(* IEC 61131-3 sources: Few-few/plc/src, 10 files *)

(* ---- DT_Tipi.st ---- *)
(*
 ============================================================================
   DT_Tipi.st  —  Tipi e enumerazioni comuni
   Software PLC manovra ascensore (geared / idraulico) — IEC 61131-3 ST
 ============================================================================
   NOTA DI SICUREZZA: questo software gestisce SOLO la logica di manovra.
   La catena di sicurezza e' cablata e indipendente (vedi schemi/).
 ============================================================================
*)

TYPE E_StatoMacchina :
(
    ST_RIPOSO       := 0,   (* cabina ferma a piano, porte chiuse *)
    ST_PRENOTATO    := 1,   (* chiamata acquisita, valuta partenza *)
    ST_CHIUDI_PORTE := 2,   (* chiusura porte prima della marcia   *)
    ST_PARTENZA     := 3,   (* sblocco freno / apertura valvola    *)
    ST_MARCIA       := 4,   (* marcia ad alta velocita'            *)
    ST_RALLENTA     := 5,   (* rallentamento verso il piano        *)
    ST_LIVELLA      := 6,   (* livellamento a bassa velocita'      *)
    ST_ARRESTO      := 7,   (* arresto e frenatura                 *)
    ST_APRI_PORTE   := 8,   (* apertura porte al piano             *)
    ST_ATTESA       := 9,   (* attesa con porte aperte             *)
    ST_REVISIONE    := 20,  (* modo ispezione uomo presente        *)
    ST_GUASTO       := 90,  (* fuori servizio per guasto           *)
    ST_EMERGENZA    := 91   (* catena sicurezza aperta             *)
) E_StatoMacchina;
END_TYPE

TYPE E_Direzione :
(
    DIR_FERMO  := 0,
    DIR_SALITA := 1,
    DIR_DISCESA := 2
) E_Direzione;
END_TYPE

(* Parametri configurabili (mappati su Modbus per il modulo WiFi).
   I valori safety-relevant (SR) restano protetti da chiave fisica. *)
TYPE ST_Parametri :
STRUCT
    (* --- non-safety (NS) --- *)
    TempoPorteAperte   : TIME := T#5S;    (* attesa porte aperte        *)
    TempoRichiusura    : TIME := T#3S;    (* dwell prima richiusura     *)
    NudgingAbilitato   : BOOL := TRUE;    (* richiusura forzata         *)
    TempoLuceOff       : TIME := T#120S;  (* spegnimento luce cabina    *)
    PianoParcheggio    : INT  := 0;       (* piano di sosta             *)
    RitardoParcheggio  : TIME := T#60S;
    GongAbilitato      : BOOL := TRUE;
    (* --- safety-relevant (SR) — modificabili solo con chiave fisica --- *)
    VelocitaIspezione  : REAL := 0.30;    (* m/s, <= 0.63 EN 81-20      *)
    VelocitaLivell     : REAL := 0.05;    (* m/s, <= 0.30               *)
    FinestraZonaPorta  : INT  := 35;      (* mm                         *)
    RelivellAbilitato  : BOOL := TRUE;
END_STRUCT
END_TYPE

(* Comandi calcolati dalla logica di posizionamento *)
TYPE ST_RichiestaCorsa :
STRUCT
    PianoTarget : INT := -1;     (* -1 = nessuna richiesta *)
    Direzione   : E_Direzione := DIR_FERMO;
    Valida      : BOOL := FALSE;
END_STRUCT
END_TYPE

(* ---- GVL_IO.st ---- *)
(*
 ============================================================================
   GVL_IO.st  —  Lista variabili globali / mappatura I/O fisica
   Software PLC manovra ascensore (geared / idraulico) — IEC 61131-3 ST
 ============================================================================
   Indirizzi %I / %Q indicativi per CPU Siemens S7-1200 1214C (DI14/DQ10)
   + moduli di espansione. Adattare alla configurazione reale.
   N. fermate di riferimento: 6 (piani 0..5).
 ============================================================================
*)

VAR_GLOBAL CONSTANT
    N_PIANI : INT := 6;   (* piani 0..5 *)
END_VAR

(* -------------------------- INGRESSI DIGITALI -------------------------- *)
VAR_GLOBAL
    (* sicurezza e modi *)
    xCatenaSicurezzaOK : BOOL AT %I0.0;   (* -KA-SIC feedback (1 = catena chiusa) *)
    xRevisione         : BOOL AT %I0.1;   (* -S-REV selettore revisione *)
    xRevSalita         : BOOL AT %I0.2;   (* -SB-REVU uomo presente su *)
    xRevDiscesa        : BOOL AT %I0.3;   (* -SB-REVD uomo presente giu *)

    (* posizione *)
    xZonaPorta1        : BOOL AT %I0.4;   (* -B-ZP1 *)
    xZonaPorta2        : BOOL AT %I0.5;   (* -B-ZP2 (ridondante) *)
    xRallentSalita     : BOOL AT %I0.6;   (* -B-RALL-U camma rallentamento su *)
    xRallentDiscesa    : BOOL AT %I0.7;   (* -B-RALL-D camma rallentamento giu *)
    xImpulsoPiano      : BOOL AT %I1.0;   (* -B-PIANI conteggio piani / encoder *)

    (* porte e carico *)
    xSovraccarico      : BOOL AT %I1.1;   (* -S-SOVR *)
    xFotocellula       : BOOL AT %I1.2;   (* -S-FOTO costa/barriera (1 = libero) *)
    xPortaAperta       : BOOL AT %I1.3;   (* -S-FAP finecorsa porta aperta *)
    xPortaChiusa       : BOOL AT %I1.4;   (* -S-FCP finecorsa porta chiusa *)

    (* protezioni macchina *)
    xTermicaMotore     : BOOL AT %I1.5;   (* -F-MOT 1 = ok *)
    xPressioneMin      : BOOL AT %I1.6;   (* -S-MINP solo idraulico, 1 = ok *)
    xControlloFreno    : BOOL AT %I1.7;   (* -S-FRE solo geared, 1 = freno integro *)

    (* chiamate cabina (parola, bit per piano) e chiamate piano *)
    wChiamateCabina    : WORD AT %IW2;    (* -SB-CAB-0..5 *)
    wChiamatePianoSu   : WORD AT %IW4;    (* -SB-PIA up   *)
    wChiamatePianoGiu  : WORD AT %IW6;    (* -SB-PIA down *)
END_VAR

(* --------------------------- USCITE DIGITALI -------------------------- *)
VAR_GLOBAL
    (* trazione geared *)
    xKM_Salita   : BOOL AT %Q0.0;   (* -KM-S *)
    xKM_Discesa  : BOOL AT %Q0.1;   (* -KM-D *)
    xKM_Veloce   : BOOL AT %Q0.2;   (* -KM-V alta velocita' (2V) *)
    xKM_Lento    : BOOL AT %Q0.3;   (* -KM-L bassa velocita' (2V) *)
    xKM_Freno    : BOOL AT %Q0.4;   (* -KM-FRE comando freno *)

    (* idraulico *)
    xKM_Pompa    : BOOL AT %Q0.5;   (* -KM-P linea pompa *)
    xKM_Stella   : BOOL AT %Q0.6;   (* -KM-Y *)
    xKM_Triangolo: BOOL AT %Q0.7;   (* -KM-Δ *)
    xEV_Salita   : BOOL AT %Q1.0;   (* -EV-S valvola salita *)
    xEV_Discesa  : BOOL AT %Q1.1;   (* -EV-D valvola discesa *)

    (* porte e segnalazioni *)
    xKM_ApriPorte  : BOOL AT %Q1.2; (* -KM-APRE *)
    xKM_ChiudiPorte: BOOL AT %Q1.3; (* -KM-CHIU *)
    xGong          : BOOL AT %Q1.4; (* -H-GONG *)
    xFuoriServizio : BOOL AT %Q1.5; (* -H-OOS *)
    wDisplayPos    : WORD AT %QW2;  (* -H-POS posizione cabina *)
    wFrecceDir     : WORD AT %QW4;  (* -H-DIR direzione *)
END_VAR

(* ------------------------- VARIABILI INTERNE -------------------------- *)
VAR_GLOBAL
    Par           : ST_Parametri;        (* parametri (anche via Modbus/WiFi) *)
    iPianoCorrente: INT := 0;            (* piano corrente stimato *)
    eDirezione    : E_Direzione := DIR_FERMO;
    eStato        : E_StatoMacchina := ST_RIPOSO;
    awChiamate    : ARRAY[0..5] OF BOOL; (* registro chiamate consolidato *)
END_VAR

(* ---- FC_Util.st ---- *)
(*
 ============================================================================
   FC_Util.st  —  Funzioni di utilita' per la mappatura Modbus dei parametri
 ============================================================================
   Conversioni registro<->valore scalato e secondi<->TIME.
   Usate da FB_ParametriModbus.st.
 ============================================================================
*)

(* Registro WORD (intero scalato) -> valore reale fisico *)
FUNCTION RegToReal : REAL
VAR_INPUT
    w     : WORD;
    scale : REAL;
END_VAR
    RegToReal := INT_TO_REAL(WORD_TO_INT(w)) / scale;
END_FUNCTION

(* Valore reale fisico -> registro WORD (intero scalato, arrotondato) *)
FUNCTION RealToReg : WORD
VAR_INPUT
    v     : REAL;
    scale : REAL;
END_VAR
    RealToReg := INT_TO_WORD(REAL_TO_INT(v * scale));
END_FUNCTION

(* Secondi (REAL) -> TIME *)
FUNCTION SecToTime : TIME
VAR_INPUT
    s : REAL;
END_VAR
    SecToTime := DINT_TO_TIME(REAL_TO_DINT(s * 1000.0));
END_FUNCTION

(* TIME -> secondi (REAL) *)
FUNCTION TimeToSec : REAL
VAR_INPUT
    t : TIME;
END_VAR
    TimeToSec := DINT_TO_REAL(TIME_TO_DINT(t)) / 1000.0;
END_FUNCTION

(* ---- FB_AllarmeEmergenza.st ---- *)
(*
 ============================================================================
   FB_AllarmeEmergenza.st  —  Sistema di allarme e comunicazione bidirezionale
                              EN 81-28:2022
 ============================================================================
   Gestisce:
   - filtro temporale sul pulsante di allarme (evita attivazioni accidentali);
   - registrazione allarme e avvio del combinatore (autodialer GSM/PSTN);
   - segnalazioni in cabina: pittogramma GIALLO (allarme inviato) e VERDE
     (collegamento col servizio di soccorso stabilito) — EN 81-28 §4.2;
   - test automatico periodico (>= ogni 3 giorni) di linea e batteria;
   - rilevazione guasto (batteria/linea) e reset da parte del tecnico.

   NB: la comunicazione vocale e l'autonomia batteria (>= 1 h) sono garantite
   dall'unita' di comunicazione certificata; qui se ne gestisce la logica di
   attivazione, segnalazione e supervisione.
 ============================================================================
*)

FUNCTION_BLOCK FB_AllarmeEmergenza
VAR_INPUT
    xPulsanteAllarme : BOOL;   (* pulsante di allarme in cabina *)
    xUnitaCommOk     : BOOL;   (* combinatore/linea telefonica ok *)
    xBatteriaOk      : BOOL;   (* batteria del sistema di allarme ok *)
    xRiscontroOper   : BOOL;   (* il servizio di soccorso ha preso in carico *)
    xResetTecnico    : BOOL;   (* reset dopo liberazione passeggero *)
    rTempoFiltro     : REAL;   (* s, filtro pressione pulsante (es. 3 s) *)
END_VAR
VAR_OUTPUT
    xAllarmeRegistrato   : BOOL;  (* pittogramma GIALLO: allarme inviato *)
    xComunicazioneAttiva : BOOL;  (* pittogramma VERDE: collegamento stabilito *)
    xAvviaCombinatore    : BOOL;  (* comando avvio chiamata *)
    xTestInCorso         : BOOL;  (* test periodico in esecuzione *)
    xGuastoAllarme       : BOOL;  (* batteria/linea KO o test fallito *)
END_VAR
VAR
    tonFiltro  : TON;
    tonTest    : TON;     (* periodo test (72 h) *)
    tonTestDur : TON;     (* durata test *)
END_VAR

(* --- filtro pressione pulsante: registra l'allarme solo se mantenuto --- *)
tonFiltro(IN := xPulsanteAllarme, PT := SecToTime(rTempoFiltro));
IF tonFiltro.Q THEN
    xAllarmeRegistrato := TRUE;   (* latch fino al reset tecnico *)
END_IF

(* --- reset da parte del tecnico (passeggero liberato) --- *)
IF xResetTecnico THEN
    xAllarmeRegistrato   := FALSE;
    xComunicazioneAttiva := FALSE;
END_IF

(* --- avvio combinatore finche' non e' stabilita la comunicazione --- *)
xAvviaCombinatore := xAllarmeRegistrato AND NOT xComunicazioneAttiva;

(* --- collegamento stabilito quando il soccorso prende in carico --- *)
IF xAllarmeRegistrato AND xRiscontroOper THEN
    xComunicazioneAttiva := TRUE;
END_IF

(* --- test automatico periodico ogni 72 h (EN 81-28) --- *)
tonTest(IN := NOT tonTest.Q, PT := T#72H);   (* impulso periodico *)
IF tonTest.Q THEN
    xTestInCorso := TRUE;
END_IF
tonTestDur(IN := xTestInCorso, PT := T#30S);
IF tonTestDur.Q THEN
    xTestInCorso := FALSE;
END_IF

(* --- guasto: batteria/linea KO, oppure test con esito negativo --- *)
xGuastoAllarme := (NOT xBatteriaOk) OR (NOT xUnitaCommOk);

END_FUNCTION_BLOCK

(* ---- FB_CatenaSicurezza.st ---- *)
(*
 ============================================================================
   FB_CatenaSicurezza.st  —  Monitoraggio (NON sostituzione) della sicurezza
 ============================================================================
   Il PLC LEGGE lo stato della catena di sicurezza cablata e delle protezioni
   macchina per gestire la manovra in modo coerente. L'ARRESTO di sicurezza e'
   garantito dall'hardware (relè -KA-SIC + contattori), non da questo codice.
 ============================================================================
*)

FUNCTION_BLOCK FB_CatenaSicurezza
VAR_INPUT
    xCatenaOK       : BOOL;   (* feedback relè sicurezza -KA-SIC *)
    xTermica        : BOOL;   (* -F-MOT 1 = ok *)
    xPressioneMin   : BOOL;   (* idraulico: 1 = ok; geared: forzare TRUE *)
    xControlloFreno : BOOL;   (* geared: 1 = freno integro; idraulico: TRUE *)
    xZonaPorta1     : BOOL;
    xZonaPorta2     : BOOL;
    xConsensoFreno  : BOOL;   (* il freno e' attualmente comandato? *)
END_VAR
VAR_OUTPUT
    xConsensoMarcia : BOOL;   (* TRUE = condizioni ok per muovere la cabina *)
    xEmergenza      : BOOL;   (* catena aperta -> fermo immediato manovra *)
    xGuasto         : BOOL;   (* guasto protezioni -> fuori servizio *)
    xInZonaPorta    : BOOL;   (* zona di livellamento valida (ridondante) *)
    xDiscordanzaZP  : BOOL;   (* discordanza sensori zona porta *)
END_VAR
VAR
    tonDiscordanza : TON;     (* tolleranza temporale discordanza ZP *)
    tonFreno       : TON;     (* controllo coerenza freno *)
END_VAR

(* --- catena di sicurezza --- *)
xEmergenza := NOT xCatenaOK;

(* --- guasto protezioni macchina (termica / pressione) --- *)
xGuasto := (NOT xTermica) OR (NOT xPressioneMin);

(* --- zona porta ridondante: validi solo se concordi --- *)
xInZonaPorta := xZonaPorta1 AND xZonaPorta2;

(* discordanza tollerata per breve transitorio, poi guasto *)
tonDiscordanza(IN := (xZonaPorta1 XOR xZonaPorta2), PT := T#500MS);
xDiscordanzaZP := tonDiscordanza.Q;
IF xDiscordanzaZP THEN
    xGuasto := TRUE;
END_IF

(* --- coerenza freno (solo geared): se comandato chiuso ma il contatto
       segnala non integro entro 1s -> guasto --- *)
tonFreno(IN := (xConsensoFreno AND NOT xControlloFreno), PT := T#1S);
IF tonFreno.Q THEN
    xGuasto := TRUE;
END_IF

(* --- consenso marcia complessivo --- *)
xConsensoMarcia := xCatenaOK AND xTermica AND xPressioneMin
                   AND NOT xGuasto AND NOT xEmergenza;

END_FUNCTION_BLOCK

(* ---- FB_GestioneChiamate.st ---- *)
(*
 ============================================================================
   FB_GestioneChiamate.st  —  Registro chiamate + selezione prossimo piano
 ============================================================================
   Logica a raccolta semplice (collettiva selettiva). Memorizza le chiamate
   di cabina e di piano e calcola il prossimo target nel senso di marcia.
 ============================================================================
*)

FUNCTION_BLOCK FB_GestioneChiamate
VAR_INPUT
    wChiamateCabina : WORD;    (* bit per piano *)
    wChiamatePiaSu  : WORD;
    wChiamatePiaGiu : WORD;
    iPianoCorrente  : INT;
    eDirezione      : E_Direzione;
    xResetTarget    : BOOL;    (* azzera target raggiunto *)
END_VAR
VAR_OUTPUT
    Richiesta       : ST_RichiestaCorsa;
    awRegistro      : ARRAY[0..5] OF BOOL;  (* chiamate attive consolidate *)
    xChiamateAttive : BOOL;
END_VAR
VAR
    i        : INT;
    iTarget  : INT := -1;
    bCabina  : ARRAY[0..5] OF BOOL;
    bSu      : ARRAY[0..5] OF BOOL;
    bGiu     : ARRAY[0..5] OF BOOL;
END_VAR

(* --- esplode le word in bit e consolida le chiamate --- *)
xChiamateAttive := FALSE;
FOR i := 0 TO 5 DO
    bCabina[i] := (wChiamateCabina AND SHL(WORD#1, INT_TO_USINT(i))) <> 0;
    bSu[i]     := (wChiamatePiaSu  AND SHL(WORD#1, INT_TO_USINT(i))) <> 0;
    bGiu[i]    := (wChiamatePiaGiu AND SHL(WORD#1, INT_TO_USINT(i))) <> 0;
    awRegistro[i] := awRegistro[i] OR bCabina[i] OR bSu[i] OR bGiu[i];
    IF awRegistro[i] THEN
        xChiamateAttive := TRUE;
    END_IF
END_FOR

(* --- cancella la chiamata del piano corrente quando vi si arriva --- *)
IF xResetTarget AND (iPianoCorrente >= 0) AND (iPianoCorrente <= 5) THEN
    awRegistro[iPianoCorrente] := FALSE;
END_IF

(* --- selezione prossimo target ---
   Priorita': prosegui nel senso di marcia finche' ci sono chiamate avanti,
   poi inverti. *)
iTarget := -1;

IF eDirezione = DIR_SALITA THEN
    FOR i := iPianoCorrente + 1 TO 5 DO
        IF awRegistro[i] AND iTarget = -1 THEN iTarget := i; END_IF
    END_FOR
    IF iTarget = -1 THEN
        FOR i := iPianoCorrente - 1 TO 0 BY -1 DO
            IF awRegistro[i] AND iTarget = -1 THEN iTarget := i; END_IF
        END_FOR
    END_IF
ELSIF eDirezione = DIR_DISCESA THEN
    FOR i := iPianoCorrente - 1 TO 0 BY -1 DO
        IF awRegistro[i] AND iTarget = -1 THEN iTarget := i; END_IF
    END_FOR
    IF iTarget = -1 THEN
        FOR i := iPianoCorrente + 1 TO 5 DO
            IF awRegistro[i] AND iTarget = -1 THEN iTarget := i; END_IF
        END_FOR
    END_IF
ELSE
    (* fermo: cerca la chiamata piu' vicina *)
    FOR i := 0 TO 5 DO
        IF awRegistro[i] AND iTarget = -1 THEN iTarget := i; END_IF
    END_FOR
END_IF

(* --- compone l'uscita --- *)
Richiesta.PianoTarget := iTarget;
Richiesta.Valida := (iTarget >= 0);
IF iTarget > iPianoCorrente THEN
    Richiesta.Direzione := DIR_SALITA;
ELSIF iTarget < iPianoCorrente AND iTarget >= 0 THEN
    Richiesta.Direzione := DIR_DISCESA;
ELSE
    Richiesta.Direzione := DIR_FERMO;
END_IF

END_FUNCTION_BLOCK

(* ---- FB_GestionePorte.st ---- *)
(*
 ============================================================================
   FB_GestionePorte.st  —  Gestione operatore porte automatiche
 ============================================================================
   Apertura/chiusura porte con fotocellula, tempo di attesa, nudging.
   La richiusura NON parte se la cabina non e' in zona di livellamento.
 ============================================================================
*)

FUNCTION_BLOCK FB_GestionePorte
VAR_INPUT
    xComandoApri    : BOOL;   (* richiesta apertura (arrivo al piano)   *)
    xRichiestaChiudi: BOOL;   (* consenso a richiudere e ripartire      *)
    xPortaAperta    : BOOL;   (* -S-FAP finecorsa porta aperta          *)
    xPortaChiusa    : BOOL;   (* -S-FCP finecorsa porta chiusa          *)
    xFotocellula    : BOOL;   (* -S-FOTO 1 = passaggio libero           *)
    xSovraccarico   : BOOL;   (* -S-SOVR 1 = sovraccarico               *)
    xInZonaPorta    : BOOL;   (* consenso movimento porte solo in zona  *)
    tAttesa         : TIME;   (* Par.TempoPorteAperte                   *)
    xNudging        : BOOL;   (* Par.NudgingAbilitato                   *)
END_VAR
VAR_OUTPUT
    xApri           : BOOL;   (* -> -KM-APRE *)
    xChiudi         : BOOL;   (* -> -KM-CHIU *)
    xPorteChiuse    : BOOL;   (* porte completamente chiuse (consenso marcia) *)
    xPorteAperte    : BOOL;
    xBloccoSovracc  : BOOL;   (* segnalazione sovraccarico: non parte *)
    xProntoChiusura : BOOL;   (* dwell trascorso: si puo' uscire da ATTESA *)
END_VAR
VAR
    tonAttesa : TON;
    xAperturaInCorso : BOOL;
END_VAR

xPorteChiuse := xPortaChiusa;
xPorteAperte := xPortaAperta;
xBloccoSovracc := xSovraccarico;

(* --- richiesta di apertura: prevale sempre (sicurezza utenza) --- *)
IF xComandoApri AND xInZonaPorta THEN
    xAperturaInCorso := TRUE;
END_IF
IF xPortaAperta THEN
    xAperturaInCorso := FALSE;
END_IF

(* --- temporizzazione attesa con porte aperte --- *)
tonAttesa(IN := xPortaAperta, PT := tAttesa);
xProntoChiusura := tonAttesa.Q;   (* dwell porte trascorso *)

(* --- decisione apertura/chiusura --- *)
xApri := FALSE;
xChiudi := FALSE;

IF NOT xInZonaPorta THEN
    (* fuori zona: porte ferme chiuse, nessun comando *)
    xApri := FALSE;
    xChiudi := FALSE;

ELSIF xAperturaInCorso OR xComandoApri THEN
    xApri := NOT xPortaAperta;

ELSIF xRichiestaChiudi AND tonAttesa.Q AND NOT xSovraccarico THEN
    (* richiusura solo dopo attesa; la fotocellula riapre *)
    IF xFotocellula OR xNudging THEN
        xChiudi := NOT xPortaChiusa;
        IF NOT xFotocellula THEN
            (* nudging: richiusura lenta a costa attiva (gestita da operatore) *)
            xChiudi := xNudging;
        END_IF
    ELSE
        (* ostacolo rilevato: riapri *)
        xApri := NOT xPortaAperta;
    END_IF
END_IF

END_FUNCTION_BLOCK

(* ---- FB_ParametriModbus.st ---- *)
(*
 ============================================================================
   FB_ParametriModbus.st  —  Interfaccia parametri PLC <-> Modbus (web)
 ============================================================================
   Il modulo WiFi (ESP32) e' Modbus MASTER; il PLC e' Modbus SLAVE con un'area
   Holding Register (awHR) mappata su questo blocco. Ogni scansione:

     - NS (reg 0..15)   : applica il valore scritto dal web, con CLAMP ai limiti
                          normativi, e riscrive il valore clampato (feedback).
     - SR (reg 20..27)  : applica SOLO se la chiave fisica -S-EN e' inserita
                          (xAbilitaParam); altrimenti RIFIUTA, riscrivendo nel
                          registro il valore corrente (il web vede il rifiuto).
     - SC/RO (reg 40..57): SOLA LETTURA — il PLC scrive stato/telemetria nei
                          registri; il web non puo' modificarli.

   Doppia barriera di sicurezza: la chiave e' verificata sia dal firmware
   (gate sul GPIO) sia qui dal PLC. I limiti EN 81-20 (es. ispezione <= 0.63
   m/s, rilivellamento <= 0.30 m/s) sono enforced lato PLC come ultima difesa.

   La sicurezza di movimento resta comunque garantita dalla catena cablata.
 ============================================================================
*)

FUNCTION_BLOCK FB_ParametriModbus
VAR_IN_OUT
    Par  : ST_Parametri;            (* parametri usati dalla manovra *)
    awHR : ARRAY[0..63] OF WORD;    (* area Holding Register (Modbus slave) *)
END_VAR
VAR_INPUT
    xAbilitaParam : BOOL;           (* -S-EN chiave abilitazione parametri SR *)
    (* --- telemetria/stato da scrivere nei registri di sola lettura --- *)
    iPosizione_mm : INT;            (* reg 50 *)
    rVelocita     : REAL;           (* reg 51 m/s *)
    rCorrente     : REAL;           (* reg 52 A *)
    iTensioneBus  : INT;            (* reg 53 V *)
    diContatore   : DINT;           (* reg 54 corse *)
    iCodiceGuasto : INT;            (* reg 55 *)
    iTempOlio     : INT;            (* reg 56 degC *)
    rPressione    : REAL;           (* reg 57 bar *)
    wStatoCatena  : WORD;           (* reg 43 bitmask *)
    wFeedbackFreno: WORD;           (* reg 44 bitmask *)
    xUcmAbilitato : BOOL;           (* reg 42 *)
    rVelNominale  : REAL;           (* reg 40 *)
    rSogliaOversp : REAL;           (* reg 41 *)
END_VAR
VAR_OUTPUT
    xSrRifiutato  : BOOL;           (* TRUE se un SR e' stato rifiutato (no chiave) *)
END_VAR

(* ====================== NON-SAFETY (clamp + feedback) ====================== *)
Par.Accelerazione   := LIMIT(0.3, RegToReal(awHR[0], 100.0), 1.2);
Par.Decelerazione   := LIMIT(0.3, RegToReal(awHR[1], 100.0), 1.2);
Par.Jerk            := LIMIT(0.5, RegToReal(awHR[2], 100.0), 2.5);
Par.VelocitaLivell  := LIMIT(0.02, RegToReal(awHR[3], 1000.0), 0.10);
Par.TempoPorteAperte:= SecToTime(LIMIT(2.0, RegToReal(awHR[4], 1.0), 20.0));
Par.TempoRichiusura := SecToTime(LIMIT(1.0, RegToReal(awHR[5], 1.0), 10.0));
Par.NudgingAbilitato:= (awHR[6] <> 0);
Par.TempoLuceOff    := SecToTime(LIMIT(30.0, RegToReal(awHR[7], 1.0), 600.0));
Par.PianoParcheggio := WORD_TO_INT(LIMIT(0, WORD_TO_INT(awHR[8]), 5));
Par.RitardoParcheggio := SecToTime(LIMIT(10.0, RegToReal(awHR[9], 1.0), 600.0));
Par.LogicaChiamate  := WORD_TO_INT(LIMIT(0, WORD_TO_INT(awHR[10]), 2));
Par.GongAbilitato   := (awHR[11] <> 0);
Par.PianoVip        := WORD_TO_INT(LIMIT(0, WORD_TO_INT(awHR[12]), 5));
Par.TempoStellaTriangolo := LIMIT(0.5, RegToReal(awHR[13], 100.0), 3.0);
Par.RitardoValvolaDiscesa:= LIMIT(0.0, RegToReal(awHR[14], 100.0), 2.0);
Par.RapportoAltaVelocita := LIMIT(0.5, RegToReal(awHR[15], 100.0), 1.0);

(* feedback del valore effettivamente applicato (clampato) *)
awHR[0]  := RealToReg(Par.Accelerazione, 100.0);
awHR[1]  := RealToReg(Par.Decelerazione, 100.0);
awHR[2]  := RealToReg(Par.Jerk, 100.0);
awHR[3]  := RealToReg(Par.VelocitaLivell, 1000.0);
awHR[4]  := RealToReg(TimeToSec(Par.TempoPorteAperte), 1.0);
awHR[5]  := RealToReg(TimeToSec(Par.TempoRichiusura), 1.0);
awHR[6]  := BOOL_TO_WORD(Par.NudgingAbilitato);
awHR[7]  := RealToReg(TimeToSec(Par.TempoLuceOff), 1.0);
awHR[8]  := INT_TO_WORD(Par.PianoParcheggio);
awHR[9]  := RealToReg(TimeToSec(Par.RitardoParcheggio), 1.0);
awHR[10] := INT_TO_WORD(Par.LogicaChiamate);
awHR[11] := BOOL_TO_WORD(Par.GongAbilitato);
awHR[12] := INT_TO_WORD(Par.PianoVip);
awHR[13] := RealToReg(Par.TempoStellaTriangolo, 100.0);
awHR[14] := RealToReg(Par.RitardoValvolaDiscesa, 100.0);
awHR[15] := RealToReg(Par.RapportoAltaVelocita, 100.0);

(* ===================== SAFETY-RELEVANT (gate chiave) ====================== *)
xSrRifiutato := FALSE;
IF xAbilitaParam THEN
    (* chiave inserita: accetta con clamp ai limiti normativi *)
    Par.RelivellAbilitato   := (awHR[20] <> 0);
    Par.FinestraZonaPorta   := WORD_TO_INT(LIMIT(10, WORD_TO_INT(awHR[21]), 80));
    Par.VelocitaIspezione   := LIMIT(0.10, RegToReal(awHR[22], 100.0), 0.63);
    Par.VelocitaRelivell    := LIMIT(0.02, RegToReal(awHR[23], 1000.0), 0.30);
    Par.VelocitaAro         := LIMIT(0.05, RegToReal(awHR[24], 100.0), 0.30);
    Par.SogliaSovracorrente := WORD_TO_INT(LIMIT(100, WORD_TO_INT(awHR[25]), 200));
    Par.RitardoFreno        := LIMIT(0.20, RegToReal(awHR[26], 1000.0), 0.80);
    Par.SogliaTempOlio      := WORD_TO_INT(LIMIT(50, WORD_TO_INT(awHR[27]), 80));
ELSE
    (* chiave assente: rifiuta qualunque scrittura SR *)
    IF (awHR[20] <> BOOL_TO_WORD(Par.RelivellAbilitato))
        OR (WORD_TO_INT(awHR[21]) <> Par.FinestraZonaPorta)
        OR (awHR[22] <> RealToReg(Par.VelocitaIspezione, 100.0))
        OR (awHR[23] <> RealToReg(Par.VelocitaRelivell, 1000.0))
        OR (awHR[24] <> RealToReg(Par.VelocitaAro, 100.0))
        OR (WORD_TO_INT(awHR[25]) <> Par.SogliaSovracorrente)
        OR (awHR[26] <> RealToReg(Par.RitardoFreno, 1000.0))
        OR (WORD_TO_INT(awHR[27]) <> Par.SogliaTempOlio) THEN
        xSrRifiutato := TRUE;
    END_IF
END_IF

(* feedback SR: riscrive sempre il valore corrente (web vede lo stato reale) *)
awHR[20] := BOOL_TO_WORD(Par.RelivellAbilitato);
awHR[21] := INT_TO_WORD(Par.FinestraZonaPorta);
awHR[22] := RealToReg(Par.VelocitaIspezione, 100.0);
awHR[23] := RealToReg(Par.VelocitaRelivell, 1000.0);
awHR[24] := RealToReg(Par.VelocitaAro, 100.0);
awHR[25] := INT_TO_WORD(Par.SogliaSovracorrente);
awHR[26] := RealToReg(Par.RitardoFreno, 1000.0);
awHR[27] := INT_TO_WORD(Par.SogliaTempOlio);

(* ===================== SOLA LETTURA (SC) e TELEMETRIA (RO) ================ *)
awHR[40] := RealToReg(rVelNominale, 100.0);
awHR[41] := RealToReg(rSogliaOversp, 100.0);
awHR[42] := BOOL_TO_WORD(xUcmAbilitato);
awHR[43] := wStatoCatena;
awHR[44] := wFeedbackFreno;

awHR[50] := INT_TO_WORD(iPosizione_mm);
awHR[51] := RealToReg(rVelocita, 100.0);
awHR[52] := RealToReg(rCorrente, 10.0);
awHR[53] := INT_TO_WORD(iTensioneBus);
awHR[54] := DINT_TO_WORD(diContatore);
awHR[55] := INT_TO_WORD(iCodiceGuasto);
awHR[56] := INT_TO_WORD(iTempOlio);
awHR[57] := RealToReg(rPressione, 10.0);

END_FUNCTION_BLOCK

(* ---- PRG_Geared.st ---- *)
(*
 ============================================================================
   PRG_Geared.st  —  Programma principale ascensore A FUNE CON ARGANO (GEARED)
 ============================================================================
   Motore a 2 velocita' (Dahlander): ALTA per la marcia, BASSA per
   avvicinamento e livellamento. Freno elettromeccanico a doppio circuito.
   Variante VVVF: sostituire la gestione -KM-V/-KM-L con i consensi inverter.

   La sicurezza e' cablata (vedi schemi/). Questo programma e' solo manovra.
 ============================================================================
*)

PROGRAM PRG_Geared
VAR
    fbSic   : FB_CatenaSicurezza;
    fbPorte : FB_GestionePorte;
    fbCall  : FB_GestioneChiamate;
    fbParam : FB_ParametriModbus;   (* interfaccia parametri web/Modbus *)
    fbAllarme : FB_AllarmeEmergenza;(* EN 81-28 allarme/comunicazione *)

    iTarget   : INT := -1;
    tonArresto: TON;
    tonGong   : TON;
    xVeloce   : BOOL;     (* richiesta alta velocita' *)
    iGuasto   : INT;
    tSostaPorte : TIME;   (* sosta porte (estesa se chiamata accessibile) *)
END_VAR

(* ------------------------------------------------------------------ *)
(* 0) PARAMETRI DA INTERFACCIA WEB (Modbus) — aggiorna Par con clamp   *)
(*    e gate a chiave per i parametri safety; pubblica la telemetria.  *)
(* ------------------------------------------------------------------ *)
IF fbSic.xEmergenza THEN iGuasto := 12;
ELSIF fbSic.xGuasto THEN iGuasto := 11;
ELSE iGuasto := 0; END_IF

fbParam(
    Par := Par, awHR := awModbusHR,
    xAbilitaParam := xAbilitaParam,
    iPosizione_mm := iPianoCorrente * 3000,
    rVelocita     := SEL(xKM_Veloce, 0.3, 1.0),
    rCorrente     := 0.0,
    iTensioneBus  := 0,
    diContatore   := diContatoreCorse,
    iCodiceGuasto := iGuasto,
    iTempOlio     := 0,
    rPressione    := 0.0,
    wStatoCatena  := SEL(fbSic.xConsensoMarcia, WORD#16#0001, WORD#16#0000),
    wFeedbackFreno:= SEL(xControlloFreno, WORD#16#0001, WORD#16#0000),
    xUcmAbilitato := TRUE,
    rVelNominale  := 1.0,
    rSogliaOversp := 1.15);

(* ------------------------------------------------------------------ *)
(* 1) MONITORAGGIO SICUREZZA                                           *)
(* ------------------------------------------------------------------ *)
fbSic(
    xCatenaOK       := xCatenaSicurezzaOK,
    xTermica        := xTermicaMotore,
    xPressioneMin   := TRUE,                 (* non applicabile su geared *)
    xControlloFreno := xControlloFreno,
    xZonaPorta1     := xZonaPorta1,
    xZonaPorta2     := xZonaPorta2,
    xConsensoFreno  := xKM_Freno);

(* ------------------------------------------------------------------ *)
(* 2) CHIAMATE E SELEZIONE TARGET                                      *)
(* ------------------------------------------------------------------ *)
fbCall(
    wChiamateCabina := wChiamateCabina,
    wChiamatePiaSu  := wChiamatePianoSu,
    wChiamatePiaGiu := wChiamatePianoGiu,
    iPianoCorrente  := iPianoCorrente,
    eDirezione      := eDirezione,
    xResetTarget    := (eStato = ST_APRI_PORTE));

(* ------------------------------------------------------------------ *)
(* 2b) ALLARME E COMUNICAZIONE DI EMERGENZA (EN 81-28)                 *)
(* ------------------------------------------------------------------ *)
fbAllarme(
    xPulsanteAllarme := xPulsanteAllarme,
    xUnitaCommOk     := xUnitaCommOk,
    xBatteriaOk      := xBatteriaAllarmeOk,
    xRiscontroOper   := xRiscontroOper,
    xResetTecnico    := xResetAllarme,
    rTempoFiltro     := Par.TempoFiltroAllarme);
xAllarmeRegistrato   := fbAllarme.xAllarmeRegistrato;
xComunicazioneAttiva := fbAllarme.xComunicazioneAttiva;
xAvviaCombinatore    := fbAllarme.xAvviaCombinatore;
xGuastoAllarme       := fbAllarme.xGuastoAllarme;

(* ------------------------------------------------------------------ *)
(* 3) GESTIONE PORTE  (sosta estesa per chiamata accessibile EN 81-70) *)
(* ------------------------------------------------------------------ *)
IF xChiamataAccessibile THEN
    tSostaPorte := Par.TempoPorteAccessibile;
ELSE
    tSostaPorte := Par.TempoPorteAperte;
END_IF
fbPorte(
    xComandoApri     := (eStato = ST_APRI_PORTE) OR (eStato = ST_ATTESA),
    xRichiestaChiudi := (eStato = ST_CHIUDI_PORTE),
    xPortaAperta     := xPortaAperta,
    xPortaChiusa     := xPortaChiusa,
    xFotocellula     := xFotocellula,
    xSovraccarico    := xSovraccarico,
    xInZonaPorta     := fbSic.xInZonaPorta,
    tAttesa          := tSostaPorte,
    xNudging         := Par.NudgingAbilitato);

xKM_ApriPorte   := fbPorte.xApri;
xKM_ChiudiPorte := fbPorte.xChiudi;

(* ------------------------------------------------------------------ *)
(* 4) CONTEGGIO PIANI (semplificato a impulsi di camma)                *)
(* ------------------------------------------------------------------ *)
(* In impianto reale: usare encoder assoluto o conteggio impulsi con
   reset ai piani estremi. Qui aggiornato all'arresto in zona porta. *)
IF eStato = ST_LIVELLA AND fbSic.xInZonaPorta THEN
    iPianoCorrente := iTarget;
END_IF

(* ------------------------------------------------------------------ *)
(* 5) MACCHINA A STATI                                                 *)
(* ------------------------------------------------------------------ *)

(* --- gestione modi prioritari --- *)
IF fbSic.xEmergenza THEN
    eStato := ST_EMERGENZA;
ELSIF fbSic.xGuasto THEN
    eStato := ST_GUASTO;
ELSIF xRevisione THEN
    eStato := ST_REVISIONE;
END_IF

CASE eStato OF

    ST_RIPOSO:
        (* tutto fermo, freno chiuso, porte chiuse *)
        xKM_Salita := FALSE; xKM_Discesa := FALSE;
        xKM_Veloce := FALSE; xKM_Lento := FALSE;
        xKM_Freno  := FALSE;   (* freno serrato *)
        eDirezione := DIR_FERMO;
        IF fbCall.Richiesta.Valida AND fbSic.xConsensoMarcia THEN
            iTarget := fbCall.Richiesta.PianoTarget;
            IF iTarget = iPianoCorrente THEN
                eStato := ST_APRI_PORTE;        (* gia' al piano: apri *)
            ELSIF NOT xSovraccarico THEN
                eStato := ST_CHIUDI_PORTE;      (* sovraccarico: non parte *)
            END_IF
        END_IF

    ST_CHIUDI_PORTE:
        xKM_ChiudiPorte := TRUE;
        IF fbPorte.xPorteChiuse THEN
            IF fbCall.Richiesta.Valida AND NOT xSovraccarico THEN
                iTarget := fbCall.Richiesta.PianoTarget;
                eDirezione := fbCall.Richiesta.Direzione;
                eStato := ST_PARTENZA;
            ELSE
                (* nessun target o sovraccarico: richiusura verso riposo *)
                eStato := ST_RIPOSO;
            END_IF
        END_IF

    ST_PARTENZA:
        IF fbSic.xConsensoMarcia AND fbPorte.xPorteChiuse THEN
            (* applica direzione + bassa velocita', poi sblocca freno *)
            xKM_Salita  := (eDirezione = DIR_SALITA);
            xKM_Discesa := (eDirezione = DIR_DISCESA);
            xKM_Lento   := TRUE;
            xKM_Freno   := TRUE;   (* sblocca freno *)
            eStato := ST_MARCIA;
        ELSE
            eStato := ST_ARRESTO;
        END_IF

    ST_MARCIA:
        (* passa ad alta velocita' se distanza sufficiente *)
        xVeloce := (ABS(iTarget - iPianoCorrente) >= 1)
                   AND NOT xRallentSalita AND NOT xRallentDiscesa;
        xKM_Veloce := xVeloce;
        xKM_Lento  := NOT xVeloce;
        (* rilevazione camma di rallentamento del piano target *)
        IF (eDirezione = DIR_SALITA AND xRallentSalita)
           OR (eDirezione = DIR_DISCESA AND xRallentDiscesa) THEN
            eStato := ST_RALLENTA;
        END_IF
        IF NOT fbSic.xConsensoMarcia THEN eStato := ST_ARRESTO; END_IF

    ST_RALLENTA:
        xKM_Veloce := FALSE;
        xKM_Lento  := TRUE;       (* bassa velocita' di avvicinamento *)
        IF fbSic.xInZonaPorta THEN
            eStato := ST_LIVELLA;
        END_IF
        IF NOT fbSic.xConsensoMarcia THEN eStato := ST_ARRESTO; END_IF

    ST_LIVELLA:
        xKM_Lento := TRUE;        (* livellamento fine in zona porta *)
        IF fbSic.xInZonaPorta THEN
            eStato := ST_ARRESTO;
        END_IF

    ST_ARRESTO:
        (* serra il freno PRIMA di togliere i contattori di marcia *)
        xKM_Freno  := FALSE;
        tonArresto(IN := TRUE, PT := T#400MS);
        IF tonArresto.Q THEN
            xKM_Salita := FALSE; xKM_Discesa := FALSE;
            xKM_Veloce := FALSE; xKM_Lento := FALSE;
            tonArresto(IN := FALSE);
            diContatoreCorse := diContatoreCorse + 1;   (* telemetria corse *)
            eStato := ST_APRI_PORTE;
        END_IF

    ST_APRI_PORTE:
        tonGong(IN := TRUE, PT := T#300MS);
        xGong := Par.GongAbilitato AND tonGong.Q;
        IF fbPorte.xPorteAperte THEN
            tonGong(IN := FALSE);
            eStato := ST_ATTESA;
        END_IF

    ST_ATTESA:
        (* mantiene le porte aperte per il tempo di sosta (dwell, esteso se
           chiamata accessibile EN 81-70); esce solo a dwell trascorso *)
        IF fbPorte.xProntoChiusura THEN
            eStato := ST_CHIUDI_PORTE;
        END_IF

    ST_REVISIONE:
        (* uomo presente, solo bassa velocita', porte non automatiche *)
        xKM_Veloce := FALSE;
        xKM_ApriPorte := FALSE; xKM_ChiudiPorte := FALSE;
        xKM_Salita  := xRevSalita AND NOT xRevDiscesa AND fbSic.xConsensoMarcia;
        xKM_Discesa := xRevDiscesa AND NOT xRevSalita AND fbSic.xConsensoMarcia;
        xKM_Lento   := xKM_Salita OR xKM_Discesa;
        xKM_Freno   := xKM_Lento;
        IF NOT xRevisione THEN eStato := ST_RIPOSO; END_IF

    ST_GUASTO:
        xKM_Salita := FALSE; xKM_Discesa := FALSE;
        xKM_Veloce := FALSE; xKM_Lento := FALSE;
        xKM_Freno  := FALSE;
        xFuoriServizio := TRUE;
        IF NOT fbSic.xGuasto AND NOT xRevisione THEN
            xFuoriServizio := FALSE;
            eStato := ST_RIPOSO;
        END_IF

    ST_EMERGENZA:
        (* catena aperta: l'hardware ha gia' tolto potenza. Allinea uscite. *)
        xKM_Salita := FALSE; xKM_Discesa := FALSE;
        xKM_Veloce := FALSE; xKM_Lento := FALSE;
        xKM_Freno  := FALSE;
        xFuoriServizio := TRUE;
        IF NOT fbSic.xEmergenza THEN
            xFuoriServizio := FALSE;
            eStato := ST_RIPOSO;
        END_IF

END_CASE

(* uscite di segnalazione comuni *)
wDisplayPos := INT_TO_WORD(iPianoCorrente);
CASE eDirezione OF
    DIR_SALITA:  wFrecceDir := 1;
    DIR_DISCESA: wFrecceDir := 2;
ELSE
    wFrecceDir := 0;
END_CASE

END_PROGRAM

(* ---- PRG_Idraulico.st ---- *)
(*
 ============================================================================
   PRG_Idraulico.st  —  Programma principale ascensore IDRAULICO
 ============================================================================
   SALITA  : avvio pompa (stella-triangolo) + valvola di salita -EV-S.
   DISCESA : per gravita' aprendo la valvola di discesa -EV-D (pompa ferma).
   Livellamento e anti-deriva (re-livellamento) in zona porta.
   Discesa di emergenza a uomo presente: gestione/segnalazione (non-safety).

   La sicurezza e' cablata (vedi schemi/). Questo programma e' solo manovra.
 ============================================================================
*)

PROGRAM PRG_Idraulico
VAR
    fbSic   : FB_CatenaSicurezza;
    fbPorte : FB_GestionePorte;
    fbCall  : FB_GestioneChiamate;

    iTarget    : INT := -1;
    tonStella  : TON;     (* tempo avviamento in stella *)
    tonGong    : TON;
    tonRelivel : TON;     (* ritardo intervento anti-deriva *)
    xPompaOn   : BOOL;
END_VAR

(* ------------------------------------------------------------------ *)
(* 1) MONITORAGGIO SICUREZZA (include pressione minima)                *)
(* ------------------------------------------------------------------ *)
fbSic(
    xCatenaOK       := xCatenaSicurezzaOK,
    xTermica        := xTermicaMotore,
    xPressioneMin   := xPressioneMin,
    xControlloFreno := TRUE,                 (* non applicabile su idraulico *)
    xZonaPorta1     := xZonaPorta1,
    xZonaPorta2     := xZonaPorta2,
    xConsensoFreno  := FALSE);

(* ------------------------------------------------------------------ *)
(* 2) CHIAMATE E TARGET                                                 *)
(* ------------------------------------------------------------------ *)
fbCall(
    wChiamateCabina := wChiamateCabina,
    wChiamatePiaSu  := wChiamatePianoSu,
    wChiamatePiaGiu := wChiamatePianoGiu,
    iPianoCorrente  := iPianoCorrente,
    eDirezione      := eDirezione,
    xResetTarget    := (eStato = ST_APRI_PORTE));

(* ------------------------------------------------------------------ *)
(* 3) PORTE                                                             *)
(* ------------------------------------------------------------------ *)
fbPorte(
    xComandoApri     := (eStato = ST_APRI_PORTE) OR (eStato = ST_ATTESA),
    xRichiestaChiudi := (eStato = ST_CHIUDI_PORTE),
    xPortaAperta     := xPortaAperta,
    xPortaChiusa     := xPortaChiusa,
    xFotocellula     := xFotocellula,
    xSovraccarico    := xSovraccarico,
    xInZonaPorta     := fbSic.xInZonaPorta,
    tAttesa          := Par.TempoPorteAperte,
    xNudging         := Par.NudgingAbilitato);

xKM_ApriPorte   := fbPorte.xApri;
xKM_ChiudiPorte := fbPorte.xChiudi;

IF eStato = ST_LIVELLA AND fbSic.xInZonaPorta THEN
    iPianoCorrente := iTarget;
END_IF

(* ------------------------------------------------------------------ *)
(* 4) MACCHINA A STATI                                                  *)
(* ------------------------------------------------------------------ *)
IF fbSic.xEmergenza THEN
    eStato := ST_EMERGENZA;
ELSIF fbSic.xGuasto THEN
    eStato := ST_GUASTO;
ELSIF xRevisione THEN
    eStato := ST_REVISIONE;
END_IF

CASE eStato OF

    ST_RIPOSO:
        xKM_Pompa := FALSE; xKM_Stella := FALSE; xKM_Triangolo := FALSE;
        xEV_Salita := FALSE; xEV_Discesa := FALSE;
        eDirezione := DIR_FERMO;
        (* anti-deriva: se la cabina lascia la zona porta a fermo, re-livella *)
        tonRelivel(IN := (NOT fbSic.xInZonaPorta) AND Par.RelivellAbilitato
                          AND fbPorte.xPorteChiuse, PT := T#1S);
        IF tonRelivel.Q AND fbSic.xConsensoMarcia THEN
            iTarget := iPianoCorrente;
            eDirezione := DIR_SALITA;     (* recupero livello solo in salita *)
            eStato := ST_PARTENZA;
        ELSIF fbCall.Richiesta.Valida AND fbSic.xConsensoMarcia THEN
            iTarget := fbCall.Richiesta.PianoTarget;
            IF iTarget = iPianoCorrente THEN
                eStato := ST_APRI_PORTE;
            ELSE
                eStato := ST_CHIUDI_PORTE;
            END_IF
        END_IF

    ST_CHIUDI_PORTE:
        xKM_ChiudiPorte := TRUE;
        IF fbPorte.xPorteChiuse THEN
            eDirezione := fbCall.Richiesta.Direzione;
            eStato := ST_PARTENZA;
        END_IF

    ST_PARTENZA:
        IF NOT (fbSic.xConsensoMarcia AND fbPorte.xPorteChiuse) THEN
            eStato := ST_ARRESTO;
        ELSIF eDirezione = DIR_SALITA THEN
            (* avvio pompa in stella, poi triangolo, poi apri valvola salita *)
            xKM_Pompa := TRUE;
            xKM_Stella := TRUE;
            tonStella(IN := TRUE, PT := T#1S500MS);
            IF tonStella.Q THEN
                xKM_Stella := FALSE;
                xKM_Triangolo := TRUE;
                xEV_Salita := TRUE;
                tonStella(IN := FALSE);
                eStato := ST_MARCIA;
            END_IF
        ELSE
            (* discesa: solo valvola, pompa ferma *)
            xKM_Pompa := FALSE; xKM_Stella := FALSE; xKM_Triangolo := FALSE;
            xEV_Discesa := TRUE;
            eStato := ST_MARCIA;
        END_IF

    ST_MARCIA:
        (* in idraulico la velocita' e' regolata dalle valvole;
           rallenta all'arrivo della camma del piano target *)
        IF (eDirezione = DIR_SALITA AND xRallentSalita)
           OR (eDirezione = DIR_DISCESA AND xRallentDiscesa) THEN
            eStato := ST_RALLENTA;
        END_IF
        IF NOT fbSic.xConsensoMarcia THEN eStato := ST_ARRESTO; END_IF

    ST_RALLENTA:
        (* la valvola riduce la portata -> avvicinamento lento *)
        IF fbSic.xInZonaPorta THEN
            eStato := ST_LIVELLA;
        END_IF
        IF NOT fbSic.xConsensoMarcia THEN eStato := ST_ARRESTO; END_IF

    ST_LIVELLA:
        IF fbSic.xInZonaPorta THEN
            eStato := ST_ARRESTO;
        END_IF

    ST_ARRESTO:
        (* chiudi valvole e ferma pompa; in salita la valvola chiude prima
           della pompa per evitare colpi d'ariete *)
        xEV_Salita := FALSE; xEV_Discesa := FALSE;
        xKM_Triangolo := FALSE; xKM_Stella := FALSE; xKM_Pompa := FALSE;
        eStato := ST_APRI_PORTE;

    ST_APRI_PORTE:
        tonGong(IN := TRUE, PT := T#300MS);
        xGong := Par.GongAbilitato AND tonGong.Q;
        IF fbPorte.xPorteAperte THEN
            tonGong(IN := FALSE);
            eStato := ST_ATTESA;
        END_IF

    ST_ATTESA:
        IF fbCall.xChiamateAttive THEN
            eStato := ST_CHIUDI_PORTE;
        ELSIF fbPorte.xPorteChiuse THEN
            eStato := ST_RIPOSO;
        ELSE
            eStato := ST_CHIUDI_PORTE;
        END_IF

    ST_REVISIONE:
        xKM_ApriPorte := FALSE; xKM_ChiudiPorte := FALSE;
        IF xRevSalita AND NOT xRevDiscesa AND fbSic.xConsensoMarcia THEN
            xKM_Pompa := TRUE; xKM_Triangolo := TRUE; xEV_Salita := TRUE;
        ELSIF xRevDiscesa AND NOT xRevSalita AND fbSic.xConsensoMarcia THEN
            xEV_Discesa := TRUE; xKM_Pompa := FALSE;
        ELSE
            xKM_Pompa := FALSE; xKM_Stella := FALSE; xKM_Triangolo := FALSE;
            xEV_Salita := FALSE; xEV_Discesa := FALSE;
        END_IF
        IF NOT xRevisione THEN eStato := ST_RIPOSO; END_IF

    ST_GUASTO:
        xKM_Pompa := FALSE; xKM_Stella := FALSE; xKM_Triangolo := FALSE;
        xEV_Salita := FALSE; xEV_Discesa := FALSE;
        xFuoriServizio := TRUE;
        IF NOT fbSic.xGuasto AND NOT xRevisione THEN
            xFuoriServizio := FALSE;
            eStato := ST_RIPOSO;
        END_IF

    ST_EMERGENZA:
        xKM_Pompa := FALSE; xKM_Stella := FALSE; xKM_Triangolo := FALSE;
        xEV_Salita := FALSE; xEV_Discesa := FALSE;
        xFuoriServizio := TRUE;
        IF NOT fbSic.xEmergenza THEN
            xFuoriServizio := FALSE;
            eStato := ST_RIPOSO;
        END_IF

END_CASE

wDisplayPos := INT_TO_WORD(iPianoCorrente);
CASE eDirezione OF
    DIR_SALITA:  wFrecceDir := 1;
    DIR_DISCESA: wFrecceDir := 2;
ELSE
    wFrecceDir := 0;
END_CASE

END_PROGRAM
